ABB RAPID module: TCP_mtip_tool2_nest2.mod

MODULE TCP_mtip_tool2_nest2
	! Points are read in order of declaration.
  ! Please do not change the order of points!

  LOCAL PERS robtarget pTCP_Point1:=[[89.36689,-966.4291,499.5596],[0.158489778637886,-0.631505012512207,0.732207298278809,-0.199887126684189],[-1,-2,-1,1],[9E+09,9E+09,9E+09,9E+09,9E+09,9E+09]];
	LOCAL PERS robtarget pTCP_Point2:=[[179.232,-1129.245,539.6489],[0.181109264492989,-0.653979361057281,0.730391561985016,-0.077708788216114],[-1,-2,-1,1],[9E+09,9E+09,9E+09,9E+09,9E+09,9E+09]];
	LOCAL PERS robtarget pTCP_Point3:=[[309.7089,-1306.12,533.3372],[0.207421958446503,-0.809472620487213,0.548938632011414,0.0199142564088106],[-1,-2,-1,1],[9E+09,9E+09,9E+09,9E+09,9E+09,9E+09]];
	LOCAL PERS robtarget pTCP_Point4:=[[503.5572,-1410.853,497.7834],[0.201106309890747,-0.817016661167145,0.51484614610672,0.164235979318619],[-1,-2,-1,1],[9E+09,9E+09,9E+09,9E+09,9E+09,9E+09]];
	LOCAL PERS robtarget pTCP_Point5:=[[779.8889,-1166.913,514.2722],[0.124469578266144,0.579337179660797,-0.77891880273819,-0.205332145094872],[-1,-3,0,1],[9E+09,9E+09,9E+09,9E+09,9E+09,9E+09]];
	LOCAL PERS robtarget pTCP_Point6:=[[780.4338,-933.0804,519.9691],[0.117356769740582,0.948606729507446,-0.216929838061333,-0.198277845978737],[-1,-3,0,1],[9E+09,9E+09,9E+09,9E+09,9E+09,9E+09]];
	LOCAL PERS robtarget pTCP_Point7:=[[494.1066,-883.637,583.0521],[0.102999866008759,0.893173098564148,-0.437152326107025,0.0230358112603426],[-1,-3,0,1],[9E+09,9E+09,9E+09,9E+09,9E+09,9E+09]];
	LOCAL PERS robtarget pTCP_Point8:=[[193.2502,-959.6873,547.544],[0.0856070294976234,-0.70311313867569,0.686928033828735,-0.162583023309708],[-1,-2,-1,1],[9E+09,9E+09,9E+09,9E+09,9E+09,9E+09]];

ENDMODULE
